{attribute 'qualified_only'}
{attribute 'strict'}
TYPE LogTechStatus:
(
  	STOPPED			:= 0,
   	RESETTING		:= 1,
   	READY			:= 2,
   	INITIALIZING	:= 3,
 	RUNNING			:= 4,
    STOPPING		:= 5,
   	ERROR			:= 6
);
END_TYPE

(* stored: Version 1.1.0.1, ProductVersion 3.1.4024.12
   DUT LogTechStatus: Id {6608dcd2-28f5-41d0-a5b1-8733183bf007} *)
